Fanuc KAREL source: kb00048.KL

-- PROVISIONAL review KL for V940-1; original PC SHA256 f850d8c97f3efb13e7014c42864522c0152b1d48fa3d7db0bbb185380ede0a95
-- Incomplete behavior may be omitted. Consult companion uncertainty JSON. Do not deploy.
PROGRAM KB00048
%NOLOCKGROUP
VAR
  P1 : REAL
  RESULT : REAL
BEGIN
  -- V9_ZERO_TABLE_METADATA_HINT layout=0001; no indexed target words; source/name/runtime held
  -- UNRESOLVED_PC offsets 5-16; opcodes 2E,23
  -- UNRESOLVED_PC offsets 21-36; opcodes 27,22,76,23
  -- UNRESOLVED_PC offsets 41-45; opcodes 7F
END KB00048
